(* CoDeSys 2.3 export: ATTR_TU.EXP *)

(* Data type in Diag/Parameter *)
TYPE attr_tu :
STRUCT
	NumberOfDigits_u16	: UINT;
	BargraphMaximum_u16	: UINT;
	PostCommaDigits_u16	: UINT;
	data_au8 				: ARRAY [1..2] OF USINT;
END_STRUCT
END_TYPE
